// TIA Portal V18 export
FUNCTION "AHU_Regulation" : Void   // FC60200, FBD
{ S7_Optimized_Access := 'TRUE' }
VERSION : 0.1
// stored: AutoNumber false, IsIECCheckEnabled false, SetENOAutomatically false, UDAEnableTagReadback false
   VAR_INPUT
      iUnitID : Int;   // 1=AHUFood, 2=AHUNonFood
   END_VAR
   VAR_TEMP
      FA_temp : Real;
   END_VAR
BEGIN

REGION Network 1 (SCL): Actual Room (salles area temp)
   // 0=PLC_IO, 1=LoraAvg, 2=MSensor,3 =Auto
   CASE "AHUAI".AI.cRoomTempSelect[#iUnitID] OF
       0:  // 
           "AHUAI".AI.rRoomAirTemp_Actual[#iUnitID] := "AHUAI".AI.rRoomAirTemp_PLC_AI[#iUnitID];
       1:  // 
           "AHUAI".AI.rRoomAirTemp_Actual[#iUnitID] := "AHUAI".AI.rRoomAirTemp_LoraAvg[#iUnitID];
       2: // 
           "AHUAI".AI.rRoomAirTemp_Actual[#iUnitID] := "AHUAI".AI.rRoomAirTemp_MSensor[#iUnitID];
       ELSE
           "AHUAI".AI.rRoomAirTemp_Actual[#iUnitID] := "AHUAI".AI.rRoomAirTemp_PLC_AI[#iUnitID];
   END_CASE;
END_REGION

REGION Network 2: AHUs SetPoints define
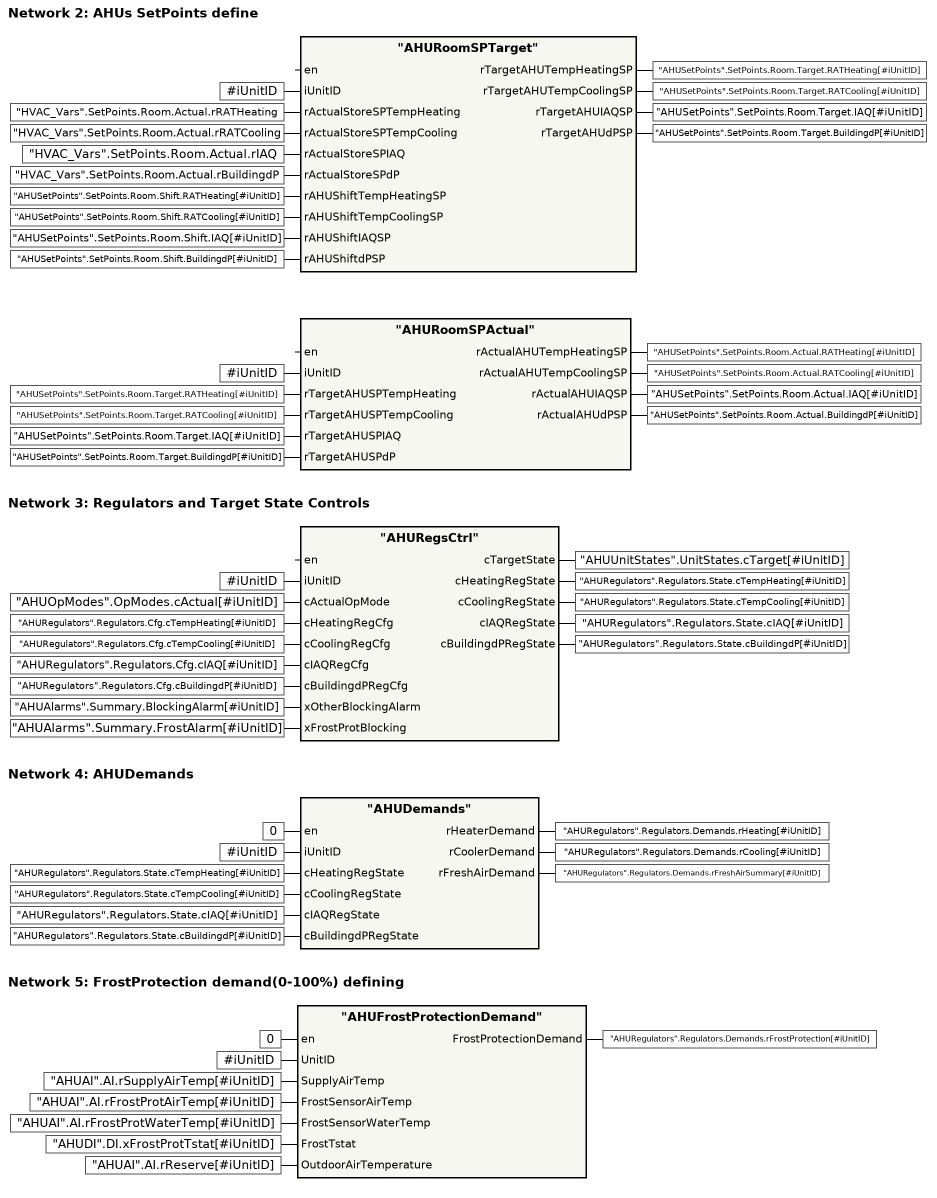
   "AHURoomSPTarget"(iUnitID := #iUnitID,
                     rActualStoreSPTempHeating := "HVAC_Vars".SetPoints.Room.Actual.rRATHeating,
                     rActualStoreSPTempCooling := "HVAC_Vars".SetPoints.Room.Actual.rRATCooling,
                     rActualStoreSPIAQ := "HVAC_Vars".SetPoints.Room.Actual.rIAQ,
                     rActualStoreSPdP := "HVAC_Vars".SetPoints.Room.Actual.rBuildingdP,
                     rAHUShiftTempHeatingSP := "AHUSetPoints".SetPoints.Room.Shift.RATHeating[#iUnitID],
                     rAHUShiftTempCoolingSP := "AHUSetPoints".SetPoints.Room.Shift.RATCooling[#iUnitID],
                     rAHUShiftIAQSP := "AHUSetPoints".SetPoints.Room.Shift.IAQ[#iUnitID],
                     rAHUShiftdPSP := "AHUSetPoints".SetPoints.Room.Shift.BuildingdP[#iUnitID],
                     rTargetAHUTempHeatingSP => "AHUSetPoints".SetPoints.Room.Target.RATHeating[#iUnitID],
                     rTargetAHUTempCoolingSP => "AHUSetPoints".SetPoints.Room.Target.RATCooling[#iUnitID],
                     rTargetAHUIAQSP => "AHUSetPoints".SetPoints.Room.Target.IAQ[#iUnitID],
                     rTargetAHUdPSP => "AHUSetPoints".SetPoints.Room.Target.BuildingdP[#iUnitID]);
   "AHURoomSPActual"(iUnitID := #iUnitID,
                     rTargetAHUSPTempHeating := "AHUSetPoints".SetPoints.Room.Target.RATHeating[#iUnitID],
                     rTargetAHUSPTempCooling := "AHUSetPoints".SetPoints.Room.Target.RATCooling[#iUnitID],
                     rTargetAHUSPIAQ := "AHUSetPoints".SetPoints.Room.Target.IAQ[#iUnitID],
                     rTargetAHUSPdP := "AHUSetPoints".SetPoints.Room.Target.BuildingdP[#iUnitID],
                     rActualAHUTempHeatingSP => "AHUSetPoints".SetPoints.Room.Actual.RATHeating[#iUnitID],
                     rActualAHUTempCoolingSP => "AHUSetPoints".SetPoints.Room.Actual.RATCooling[#iUnitID],
                     rActualAHUIAQSP => "AHUSetPoints".SetPoints.Room.Actual.IAQ[#iUnitID],
                     rActualAHUdPSP => "AHUSetPoints".SetPoints.Room.Actual.BuildingdP[#iUnitID]);
END_REGION

REGION Network 3: Regulators and Target State Controls
   "AHURegsCtrl"(iUnitID := #iUnitID,
                 cActualOpMode := "AHUOpModes".OpModes.cActual[#iUnitID],
                 cHeatingRegCfg := "AHURegulators".Regulators.Cfg.cTempHeating[#iUnitID],
                 cCoolingRegCfg := "AHURegulators".Regulators.Cfg.cTempCooling[#iUnitID],
                 cIAQRegCfg := "AHURegulators".Regulators.Cfg.cIAQ[#iUnitID],
                 cBuildingdPRegCfg := "AHURegulators".Regulators.Cfg.cBuildingdP[#iUnitID],
                 xOtherBlockingAlarm := "AHUAlarms".Summary.BlockingAlarm[#iUnitID],
                 xFrostProtBlocking := "AHUAlarms".Summary.FrostAlarm[#iUnitID],
                 cTargetState => "AHUUnitStates".UnitStates.cTarget[#iUnitID],
                 cHeatingRegState => "AHURegulators".Regulators.State.cTempHeating[#iUnitID],
                 cCoolingRegState => "AHURegulators".Regulators.State.cTempCooling[#iUnitID],
                 cIAQRegState => "AHURegulators".Regulators.State.cIAQ[#iUnitID],
                 cBuildingdPRegState => "AHURegulators".Regulators.State.cBuildingdP[#iUnitID]);
END_REGION

REGION Network 4: AHUDemands
   // Regulator State -> Demands
   IF 0 THEN
       "AHUDemands"(iUnitID := #iUnitID,
                    cHeatingRegState := "AHURegulators".Regulators.State.cTempHeating[#iUnitID],
                    cCoolingRegState := "AHURegulators".Regulators.State.cTempCooling[#iUnitID],
                    cIAQRegState := "AHURegulators".Regulators.State.cIAQ[#iUnitID],
                    cBuildingdPRegState := "AHURegulators".Regulators.State.cBuildingdP[#iUnitID],
                    rHeaterDemand => "AHURegulators".Regulators.Demands.rHeating[#iUnitID],
                    rCoolerDemand => "AHURegulators".Regulators.Demands.rCooling[#iUnitID],
                    rFreshAirDemand => "AHURegulators".Regulators.Demands.rFreshAirSummary[#iUnitID]);
   END_IF;
END_REGION

REGION Network 5: FrostProtection demand(0-100%) defining
   IF 0 THEN
       "AHUFrostProtectionDemand"(UnitID := #iUnitID,
                               SupplyAirTemp := "AHUAI".AI.rSupplyAirTemp[#iUnitID],
                               FrostSensorAirTemp := "AHUAI".AI.rFrostProtAirTemp[#iUnitID],
                               FrostSensorWaterTemp := "AHUAI".AI.rFrostProtWaterTemp[#iUnitID],
                               FrostTstat := "AHUDI".DI.xFrostProtTstat[#iUnitID],
                               OutdoorAirTemperature := "AHUAI".AI.rReserve[#iUnitID],
                               FrostProtectionDemand => "AHURegulators".Regulators.Demands.rFrostProtection[#iUnitID]);
   END_IF;
END_REGION
END_FUNCTION
